{attribute addProperty BoxType "EK1100-0000-0018"}
{attribute addProperty Id "Beckhoff_EPP5xxxEK1122Beckhoff_EPP5xxxEK1122_277DA9AB1442180.25"}
{attribute addProperty CRC "919776683"}
{attribute addProperty SizeInBites "1442"}
{attribute addProperty SizeInBytes "180.25"}
TYPE Beckhoff_EPP5xxx_36D2ADAB EXTENDS EK1100_179A0949 :
STRUCT
	{attribute addProperty Name "Beckhoff_EPP5xxxEK1122"}
	Beckhoff_EPP5xxxEK1122 : Beckhoff_EPP5xxxEK1122_277DA9AB;
END_STRUCT
END_TYPE

(* stored: Version 1.2.0.0, ProductVersion 3.1.4024.9
   DUT Beckhoff_EPP5xxx_36D2ADAB: Id {cfbed035-98f4-4b59-acf3-da193e3a046b} *)
